ABB RAPID module: Wobj_wobj_A1.mod

MODULE Wobj_wobj_A1
	! Points are read in order of declaration.
  ! Please do not change the order of points!

  LOCAL PERS robtarget pWobj_U_PointX1:=[[1393.425,-1975.612,-698.908],[0.000258766231127083,-0.727538704872131,0.686066031455994,0.000880914740264416],[-1,0,2,0],[0,9E+09,9E+09,9E+09,9E+09,9E+09]];
	LOCAL PERS robtarget pWobj_U_PointX2:=[[1557.76,-1964.564,-698.8776],[0.000256818631896749,-0.727544724941254,0.686059594154358,0.000875434139743447],[-1,0,2,0],[0,9E+09,9E+09,9E+09,9E+09,9E+09]];
	LOCAL PERS robtarget pWobj_U_PointY1:=[[1557.467,-1753.91,-698.876],[0.000259275082498789,-0.727566063404083,0.686037003993988,0.000875030178576708],[-1,0,2,0],[0,9E+09,9E+09,9E+09,9E+09,9E+09]];

ENDMODULE
